FUNCTION_BLOCK E_F_TRIG (* Boolean falling edge detection *)
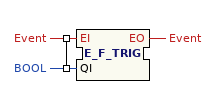
  EVENT_INPUT
    EI WITH QI; (* check for falling edge *)
  END_EVENT
  EVENT_OUTPUT
    EO; (* confirmation that an falling edge was detected *)
  END_EVENT
  VAR_INPUT
    QI : BOOL; (* value to check for a falling edge *)
  END_VAR
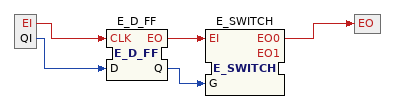
  FBS
    E_D_FF : iec61499::events::E_D_FF;
    E_SWITCH : iec61499::events::E_SWITCH;
  END_FBS
  EVENT_CONNECTIONS
    EI TO E_D_FF.CLK;
    E_D_FF.EO TO E_SWITCH.EI;
    E_SWITCH.EO0 TO EO;
  END_CONNECTIONS
  DATA_CONNECTIONS
    QI TO E_D_FF.D;
    E_D_FF.Q TO E_SWITCH.G;
  END_CONNECTIONS
END_FUNCTION_BLOCK
